PROGRAM BackgroundComm
VAR
END_VAR

HWVar.ModbusMaster();
HWVar.ModbusMaster1();

END_PROGRAM

(* stored: Version 1.1.0.1, ProductVersion 3.1.4022.18
   POU BackgroundComm: Id {40779a71-740b-4a35-a3c1-34d5abe4afe3}, SpecialFunc None *)
